TYPE ST_JointDirection :
STRUCT	
	Left 	: BOOL;
	Right	: BOOL;
END_STRUCT
END_TYPE

(* stored: Version 1.1.0.1, ProductVersion 3.1.4024.9
   DUT ST_JointDirection: Id {ca86a206-bc04-4298-be8f-9fadc8ba7dfd} *)
